MOVL C00519 BC00519 V=1000.0  +MOVJ EC00519 VJ=100.00
MOVJ C00520 BC00520 VJ=100.00  +MOVJ EC00520 VJ=100.00
'Path S3689
SFTOF3D
MOVJ C00521 BC00521 VJ=100.00  +MOVJ EC00521 VJ=100.00
MOVL C00522 BC00522 V=400.0  +MOVJ EC00522 VJ=100.00
SMOVL C00523 BC00523 V=100.0  +MOVJ EC00523
SREFP 3 C00524 BC00524  +REFP EC00524
CALL JOB:SEARCH-R1-S13D
SET P022 P006
SFTON3D P022
SMOVL C00525 BC00525 V=100.0  +MOVJ EC00525
SREFP 3 C00526 BC00526  +REFP EC00526
CALL JOB:SEARCH-R1-S13D
SET P022 P006
SFTON3D P022
SMOVL C00527 BC00527 V=250.0  +MOVJ EC00527
SFTOF3D
SMOVL C00528 BC00528 V=1000.0  +MOVJ EC00528
SMOVL C00529 BC00529 V=1000.0  +MOVJ EC00529
SMOVL C00530 BC00530 V=1000.0  +MOVJ EC00530
SMOVL C00531 BC00531 V=333.3  +MOVJ EC00531
SREFP 3 C00532 BC00532  +REFP EC00532
CALL JOB:SEARCH-R1-S13D
SET P060 P006
SFTON3D P060
SMOVL C00533 BC00533 V=166.7  +MOVJ EC00533
SMOVL C00534 BC00534 V=166.7  +MOVJ EC00534
SREFP 3 C00535 BC00535  +REFP EC00535
CALL JOB:SEARCH-R1-S13D
SET P060 P006
SFTON3D P060
SMOVL C00536 BC00536 V=166.7  +MOVJ EC00536
MOVJ C00537 BC00537 VJ=15.00  +MOVJ EC00537 VJ=0.78
MOVJ C00538 BC00538 VJ=15.00  +MOVJ EC00538 VJ=15.00
SMOVL C00539 BC00539 V=166.7  +MOVJ EC00539
SREFP 3 C00540 BC00540  +REFP EC00540
CALL JOB:SEARCH-R1-S13D
SET P060 P006
SFTON3D P060
SMOVL C00541 BC00541 V=416.7  +MOVJ EC00541
SFTOF3D
SMOVL C00542 BC00542 V=416.7  +MOVJ EC00542
SMOVL C00543 BC00543 V=416.7  +MOVJ EC00543
SREFP 3 C00544 BC00544  +REFP EC00544
CALL JOB:SEARCH-R1-S13D
SET P061 P006
SFTON3D P061
SMOVL C00545 BC00545 V=166.7  +MOVJ EC00545
SREFP 3 C00546 BC00546  +REFP EC00546
CALL JOB:SEARCH-R1-S13D
SET P061 P006
SFTON3D P061
SMOVL C00547 BC00547 V=500.0  +MOVJ EC00547
SMOVL C00548 BC00548 V=500.0  +MOVJ EC00548
SMOVL C00549 BC00549 V=1000.0  +MOVJ EC00549
MOVJ C00550 BC00550 VJ=100.00  +MOVJ EC00550 VJ=100.00
MOVJ C00551 BC00551 VJ=100.00  +MOVJ EC00551 VJ=100.00
MOVJ C00552 BC00552 VJ=100.00  +MOVJ EC00552 VJ=100.00
'Path S3690
SFTOF3D
MOVJ C00553 BC00553 VJ=100.00  +MOVJ EC00553 VJ=100.00
MOVL C00554 BC00554 V=400.0  +MOVJ EC00554 VJ=100.00
SMOVL C00555 BC00555 V=100.0  +MOVJ EC00555
SREFP 3 C00556 BC00556  +REFP EC00556
CALL JOB:SEARCH-R1-S13D
SET P021 P006
SFTON3D P021
SMOVL C00557 BC00557 V=100.0  +MOVJ EC00557
SREFP 3 C00558 BC00558  +REFP EC00558
CALL JOB:SEARCH-R1-S13D
SET P021 P006
SFTON3D P021
SMOVL C00559 BC00559 V=100.0  +MOVJ EC00559
SFTOF3D
MOVL C00560 BC00560 V=400.0  +MOVJ EC00560 VJ=100.00
SFTON3D P021
SMOVL C00561 BC00561 V=166.7 PL=0  +MOVJ EC00561
SREFP 1 C00562 BC00562  +REFP EC00562
SREFP 2 C00563 BC00563  +REFP EC00563
MACRO1 MJ#(0) ARGF9
ARCON
SMOVL C00564 BC00564 V=12.5  +MOVJ EC00564
SMOVL C00565 BC00565 V=12.5  +MOVJ EC00565
ARCOF
SFTOF3D
MOVL C00566 BC00566 V=400.0  +MOVJ EC00566 VJ=100.00
MOVL C00567 BC00567 V=1000.0  +MOVJ EC00567 VJ=100.00
MOVJ C00568 BC00568 VJ=100.00  +MOVJ EC00568 VJ=100.00
MOVJ C00569 BC00569 VJ=100.00  +MOVJ EC00569 VJ=100.00
MOVJ C00570 BC00570 VJ=100.00  +MOVJ EC00570 VJ=100.00
'2
'Path W3693
SFTOF3D
MOVJ C00571 BC00571 VJ=100.00  +MOVJ EC00571 VJ=100.00
MACRO1 MJ#(0) ARGF6
SFTON3D P060
SMOVL C00572 BC00572 V=166.7  +MOVJ EC00572
ARCON
SMOVL C00573 BC00573 V=8.3  +MOVJ EC00573
SMOVL C00574 BC00574 V=8.3  +MOVJ EC00574
SMOVL C00575 BC00575 V=8.3  +MOVJ EC00575
ARCOF
SMOVL C00576 BC00576 V=166.7  +MOVJ EC00576
SMOVL C00577 BC00577 V=333.3  +MOVJ EC00577
MACRO1 MJ#(0) ARGF14
SFTON3D P061
SMOVL C00578 BC00578 V=166.7  +MOVJ EC00578
ARCON
SMOVL C00579 BC00579 V=10.0  +MOVJ EC00579
ARCOF
SFTOF3D
SMOVL C00580 BC00580 V=416.7  +MOVJ EC00580
MOVJ C00581 BC00581 VJ=100.00  +MOVJ EC00581 VJ=25.00
MOVL C00582 BC00582 V=400.0  +MOVJ EC00582 VJ=100.00
SFTON3D P023
SMOVL C00583 BC00583 V=166.7 PL=0  +MOVJ EC00583
SREFP 1 C00584 BC00584  +REFP EC00584
SREFP 2 C00585 BC00585  +REFP EC00585
MACRO1 MJ#(0) ARGF9
ARCON
SMOVL C00586 BC00586 V=11.7  +MOVJ EC00586
ARCOF
SFTOF3D
MOVL C00587 BC00587 V=400.0  +MOVJ EC00587 VJ=100.00
MOVL C00588 BC00588 V=1000.0  +MOVJ EC00588 VJ=100.00
'Path W3694
SFTOF3D
MOVJ C00589 BC00589 VJ=100.00  +MOVJ EC00589 VJ=100.00
MOVL C00590 BC00590 V=400.0  +MOVJ EC00590 VJ=100.00
SFTON3D P023
SMOVL C00591 BC00591 V=166.7 PL=0  +MOVJ EC00591
SREFP 1 C00592 BC00592  +REFP EC00592
SREFP 2 C00593 BC00593  +REFP EC00593
ARCON
SMOVL C00594 BC00594 V=11.7  +MOVJ EC00594
ARCOF
SFTOF3D
MOVL C00595 BC00595 V=400.0  +MOVJ EC00595 VJ=100.00
MOVL C00596 BC00596 V=1000.0  +MOVJ EC00596 VJ=100.00
MOVJ C00597 BC00597 VJ=100.00  +MOVJ EC00597 VJ=100.00
MOVJ C00598 BC00598 VJ=100.00  +MOVJ EC00598 VJ=100.00
MOVJ C00599 BC00599 VJ=100.00  +MOVJ EC00599 VJ=100.00
MOVJ C00600 BC00600 VJ=100.00  +MOVJ EC00600 VJ=100.00
SFTOF3D
MOVJ C00601 BC00601 VJ=100.00  +MOVJ EC00601 VJ=100.00
SFTOF3D
MOVJ C00602 BC00602 VJ=100.00  +MOVJ EC00602 VJ=100.00
MOVL C00603 BC00603 V=666.7  +MOVJ EC00603 VJ=100.00
SFTON3D P021
MACRO1 MJ#(0) ARGF9
SMOVL C00604 BC00604 V=166.7 PL=0  +MOVJ EC00604
SREFP 1 C00605 BC00605  +REFP EC00605
SREFP 2 C00606 BC00606  +REFP EC00606
ARCON
SMOVL C00607 BC00607 V=11.7  +MOVJ EC00607
ARCOF
SFTOF3D
MOVL C00608 BC00608 V=400.0  +MOVJ EC00608 VJ=100.00
MOVL C00609 BC00609 V=1000.0  +MOVJ EC00609 VJ=100.00
MOVJ C00610 BC00610 VJ=100.00  +MOVJ EC00610 VJ=100.00
MOVJ C00611 BC00611 VJ=100.00  +MOVJ EC00611 VJ=100.00
MOVJ C00612 BC00612 VJ=100.00  +MOVJ EC00612 VJ=100.00
MOVJ C00613 BC00613 VJ=100.00  +MOVJ EC00613 VJ=100.00
MOVJ C00614 BC00614 VJ=100.00  +MOVJ EC00614 VJ=100.00
'Path W3697
SFTOF3D
MOVJ C00615 BC00615 VJ=100.00  +MOVJ EC00615 VJ=100.00
MOVL C00616 BC00616 V=666.7  +MOVJ EC00616 VJ=100.00
SFTON3D P023
SMOVL C00617 BC00617 V=133.3 PL=0  +MOVJ EC00617
SREFP 1 C00618 BC00618  +REFP EC00618
SREFP 2 C00619 BC00619  +REFP EC00619
ARCON
SMOVL C00620 BC00620 V=11.7  +MOVJ EC00620
ARCOF
MOVL C00621 BC00621 V=400.0  +MOVJ EC00621 VJ=100.00
MOVL C00622 BC00622 V=1000.0  +MOVJ EC00622 VJ=100.00
'Path W3698
SFTOF3D
MOVJ C00623 BC00623 VJ=100.00  +MOVJ EC00623 VJ=100.00
MOVL C00624 BC00624 V=400.0  +MOVJ EC00624 VJ=100.00
SFTON3D P023
SMOVL C00625 BC00625 V=133.3 PL=0  +MOVJ EC00625
SREFP 1 C00626 BC00626  +REFP EC00626
SREFP 2 C00627 BC00627  +REFP EC00627
ARCON
SMOVL C00628 BC00628 V=11.7  +MOVJ EC00628
ARCOF
SFTOF3D
MOVL C00629 BC00629 V=400.0  +MOVJ EC00629 VJ=100.00
MOVL C00630 BC00630 V=1000.0  +MOVJ EC00630 VJ=100.00
'5
MOVJ C00631 BC00631 VJ=100.00  +MOVJ EC00631 VJ=100.00
MOVJ C00632 BC00632 VJ=100.00  +MOVJ EC00632 VJ=100.00
MOVJ C00633 BC00633 VJ=100.00  +MOVJ EC00633 VJ=100.00
SFTOF3D
MOVJ C00634 BC00634 VJ=100.00  +MOVJ EC00634 VJ=100.00
MOVL C00635 BC00635 V=400.0  +MOVJ EC00635 VJ=100.00
SFTON3D P022
SMOVL C00636 BC00636 V=133.3 PL=0  +MOVJ EC00636
SREFP 1 C00637 BC00637  +REFP EC00637
SREFP 2 C00638 BC00638  +REFP EC00638
ARCON
SMOVL C00639 BC00639 V=11.7  +MOVJ EC00639
ARCOF
SFTOF3D
MOVL C00640 BC00640 V=400.0  +MOVJ EC00640 VJ=100.00
MOVL C00641 BC00641 V=1000.0  +MOVJ EC00641 VJ=100.00
'6
MOVJ C00642 BC00642 VJ=100.00  +MOVJ EC00642 VJ=100.00
MOVJ C00643 BC00643 VJ=100.00  +MOVJ EC00643 VJ=100.00
MOVJ C00644 BC00644 VJ=100.00  +MOVJ EC00644 VJ=100.00
'Path W3701
SFTOF3D
MOVJ C00645 BC00645 VJ=100.00  +MOVJ EC00645 VJ=100.00
MOVJ C00646 BC00646 VJ=100.00  +MOVJ EC00646 VJ=100.00
MOVL C00647 BC00647 V=400.0  +MOVJ EC00647 VJ=100.00
SFTON3D P023
SMOVL C00648 BC00648 V=166.7 PL=0  +MOVJ EC00648
SREFP 1 C00649 BC00649  +REFP EC00649
SREFP 2 C00650 BC00650  +REFP EC00650
ARCON
SMOVL C00651 BC00651 V=11.7  +MOVJ EC00651
ARCOF
SFTOF3D
MOVL C00652 BC00652 V=400.0  +MOVJ EC00652 VJ=100.00
MOVL C00653 BC00653 V=1000.0  +MOVJ EC00653 VJ=100.00
'Path W3702
SFTOF3D
MOVJ C00654 BC00654 VJ=100.00  +MOVJ EC00654 VJ=100.00
MOVL C00655 BC00655 V=400.0  +MOVJ EC00655 VJ=100.00
SFTON3D P023
SMOVL C00656 BC00656 V=166.7 PL=0  +MOVJ EC00656
SREFP 1 C00657 BC00657  +REFP EC00657
SREFP 2 C00658 BC00658  +REFP EC00658
ARCON
SMOVL C00659 BC00659 V=12.5  +MOVJ EC00659
ARCOF
SFTOF3D
MOVL C00660 BC00660 V=400.0  +MOVJ EC00660 VJ=100.00
MOVL C00661 BC00661 V=1000.0  +MOVJ EC00661 VJ=100.00
SFTOF3D
MOVJ C00662 BC00662 VJ=100.00  +MOVJ EC00662 VJ=100.00
MOVL C00663 BC00663 V=400.0  +MOVJ EC00663 VJ=100.00
MACRO1 MJ#(0) ARGF9
SFTON3D P022
SMOVL C00664 BC00664 V=166.7 PL=0  +MOVJ EC00664
SREFP 1 C00665 BC00665  +REFP EC00665
SREFP 2 C00666 BC00666  +REFP EC00666
ARCON
SMOVL C00667 BC00667 V=11.7  +MOVJ EC00667
ARCOF
SFTOF3D
MOVL C00668 BC00668 V=400.0  +MOVJ EC00668 VJ=100.00
MOVL C00669 BC00669 V=1000.0  +MOVJ EC00669 VJ=100.00
'8
'Path W3705
SFTOF3D
MOVJ C00670 BC00670 VJ=100.00  +MOVJ EC00670 VJ=100.00
MOVL C00671 BC00671 V=400.0  +MOVJ EC00671 VJ=100.00
SFTON3D P022
SMOVL C00672 BC00672 V=166.7 PL=0  +MOVJ EC00672
SREFP 1 C00673 BC00673  +REFP EC00673
SREFP 2 C00674 BC00674  +REFP EC00674
MACRO1 MJ#(0) ARGF14
ARCON
SMOVL C00675 BC00675 V=10.0  +MOVJ EC00675
ARCOF
SFTOF3D
MOVL C00676 BC00676 V=400.0  +MOVJ EC00676 VJ=100.00
MOVL C00677 BC00677 V=1000.0  +MOVJ EC00677 VJ=100.00
'Path W3706
SFTOF3D
MOVJ C00678 BC00678 VJ=100.00  +MOVJ EC00678 VJ=100.00
MOVL C00679 BC00679 V=400.0  +MOVJ EC00679 VJ=100.00
SFTON3D P022
SMOVL C00680 BC00680 V=166.7 PL=0  +MOVJ EC00680
SREFP 1 C00681 BC00681  +REFP EC00681
SREFP 2 C00682 BC00682  +REFP EC00682
MACRO1 MJ#(0) ARGF9
ARCON
SMOVL C00683 BC00683 V=10.8  +MOVJ EC00683
ARCOF
SFTOF3D
MOVL C00684 BC00684 V=400.0  +MOVJ EC00684 VJ=100.00
MOVL C00685 BC00685 V=1000.0  +MOVJ EC00685 VJ=100.00
END
